FUNCTION_BLOCK L3_MachineManager (* Composite Function Block Type *)
  (* Standard: 61499-2 *)
  (* Version 0.0, 2014-10-06, EQUEROL, UJI *)
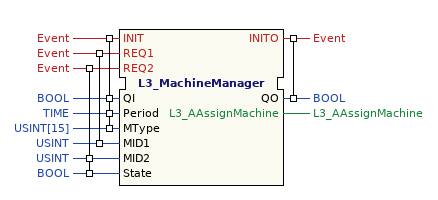
  EVENT_INPUT
    INIT WITH QI, MType, Period; (* Initialization Request *)
    REQ1 WITH MID1; (* Request to handle a released machine *)
    REQ2 WITH MID2, State; (* Request to handle a change in the operative state of a machine *)
  END_EVENT
  EVENT_OUTPUT
    INITO WITH QO; (* Initialization Confirm *)
  END_EVENT
  VAR_INPUT
    QI : BOOL; (* Input event qualifier *)
    Period : TIME := T#1000ms; (* MMCore execution period *)
    MType : ARRAY [0..14] OF USINT := [0,0,0,0,0,0,0,0,0,0,0,0,0,0,0]; (* Machine type vector *)
    MID1 : USINT; (* Machine identifier *)
    MID2 : USINT; (* Machine identifier *)
    State : BOOL; (* Machine state, true =OK, FALSE=KO *)
  END_VAR
  VAR_OUTPUT
    QO : BOOL; (* Output event qualifier *)
  END_VAR
  PLUGS
    L3_AAssignMachine : L3_AAssignMachine;
  END_PLUGS
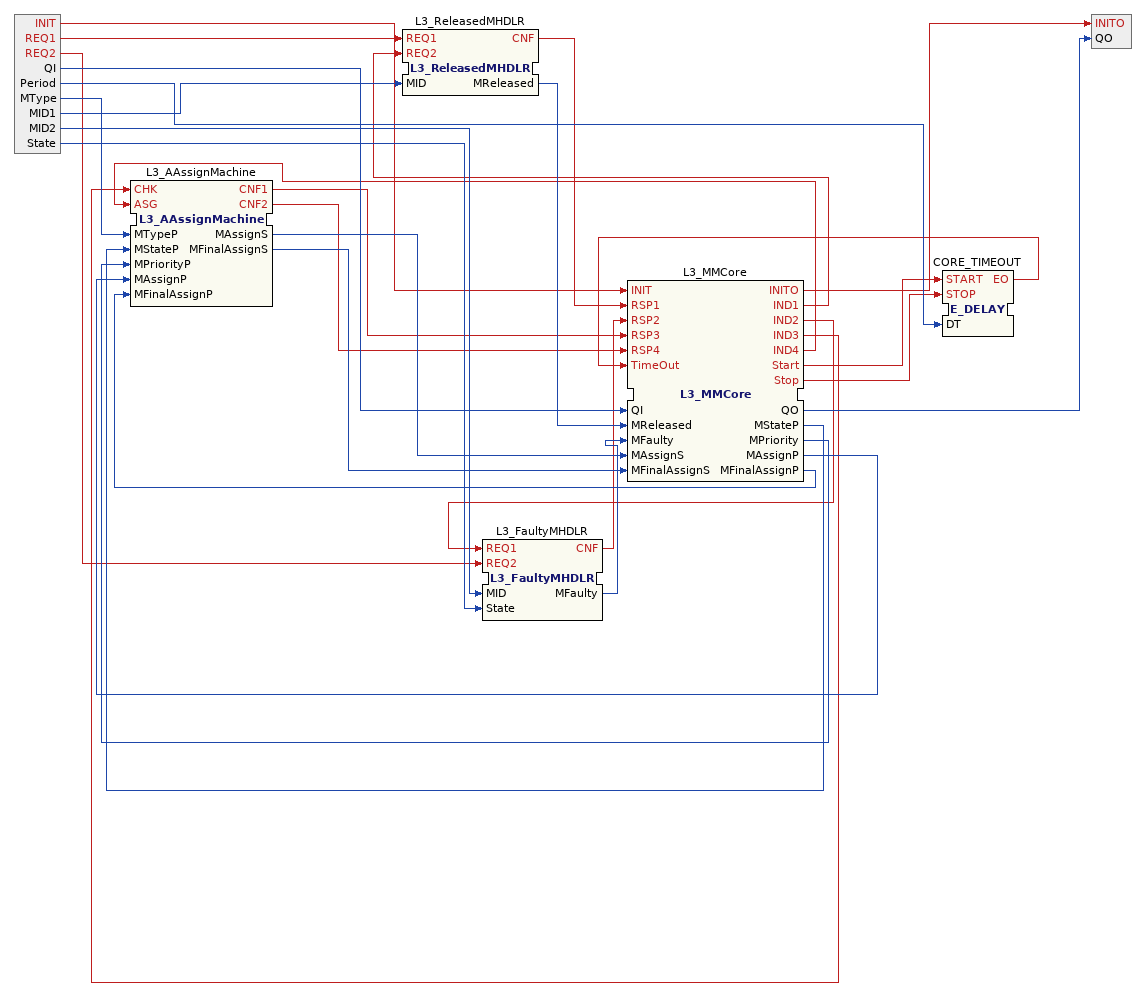
  FBS
    L3_ReleasedMHDLR : L3_ReleasedMHDLR;
    L3_FaultyMHDLR : L3_FaultyMHDLR;
    CORE_TIMEOUT : E_DELAY;
    L3_MMCore : L3_MMCore;
  END_FBS
  EVENT_CONNECTIONS
    REQ1 TO L3_ReleasedMHDLR.REQ1;
    REQ2 TO L3_FaultyMHDLR.REQ2;
    INIT TO L3_MMCore.INIT;
    L3_ReleasedMHDLR.CNF TO L3_MMCore.RSP1;
    L3_FaultyMHDLR.CNF TO L3_MMCore.RSP2;
    L3_AAssignMachine.CNF1 TO L3_MMCore.RSP3;
    L3_AAssignMachine.CNF2 TO L3_MMCore.RSP4;
    L3_MMCore.INITO TO INITO;
    L3_MMCore.IND1 TO L3_ReleasedMHDLR.REQ2;
    L3_MMCore.IND2 TO L3_FaultyMHDLR.REQ1;
    L3_MMCore.IND3 TO L3_AAssignMachine.CHK;
    L3_MMCore.IND4 TO L3_AAssignMachine.ASG;
    L3_MMCore.Start TO CORE_TIMEOUT.START;
    L3_MMCore.Stop TO CORE_TIMEOUT.STOP;
    CORE_TIMEOUT.EO TO L3_MMCore.TimeOut;
  END_CONNECTIONS
  DATA_CONNECTIONS
    MID1 TO L3_ReleasedMHDLR.MID;
    MID2 TO L3_FaultyMHDLR.MID;
    State TO L3_FaultyMHDLR.State;
    MType TO L3_AAssignMachine.MTypeP;
    QI TO L3_MMCore.QI;
    L3_ReleasedMHDLR.MReleased TO L3_MMCore.MReleased;
    L3_FaultyMHDLR.MFaulty TO L3_MMCore.MFaulty;
    L3_AAssignMachine.MAssignS TO L3_MMCore.MAssignS;
    L3_AAssignMachine.MFinalAssignS TO L3_MMCore.MFinalAssignS;
    L3_MMCore.QO TO QO;
    L3_MMCore.MStateP TO L3_AAssignMachine.MStateP;
    L3_MMCore.MPriority TO L3_AAssignMachine.MPriorityP;
    L3_MMCore.MAssignP TO L3_AAssignMachine.MAssignP;
    L3_MMCore.MFinalAssignP TO L3_AAssignMachine.MFinalAssignP;
    Period TO CORE_TIMEOUT.DT;
  END_CONNECTIONS
END_FUNCTION_BLOCK
